{attribute 'pack_mode' := '1'}
TYPE stEL3058_Channel :
STRUCT
	Status	AT %I* : stEL3058_ChannelStatus;
	Value 	AT %I* : WORD;
END_STRUCT
END_TYPE

(* stored: Version 1.1.0.1, ProductVersion 3.1.4024.4
   DUT stEL3058_Channel: Id {538fc2bc-f8d9-43cb-bcb0-ccf5729b907a} *)
